// TIA Portal project "btvn" (V14)

(* hardware
DEVICE "S7-1200 station_1"  S7-1200 Station
   slot 0: "Rack_0"  S7-1200 Rack  Rack  V1.0
   slot 1: "PLC_1"  CPU 1214C DC/DC/DC  6ES7 214-1AG40-0XB0  V4.2
*)

// ===== PLC "PLC_1"  CPU 1214C DC/DC/DC =====

VAR_GLOBAL   // PLC tag table "Default tag table"
   "button1" AT %I0.1 : Bool;
   "button2" AT %I0.2 : Bool;
   "start" AT %I0.3 : Bool;
   "red_1" AT %Q0.2 : Bool;
   "red_2" AT %Q0.3 : Bool;
   "green_1" AT %Q0.0 : Bool;
   "green2" AT %Q0.1 : Bool;
   "reset" AT %I0.4 : Bool;
   "save1" AT %M1.0 : Bool;
   "save2" AT %M1.1 : Bool;
   "Start_button_" AT %M1.2 : Bool;
   "but1" AT %M0.0 : Bool;
   "den" AT %M0.1 : Bool;
END_VAR

ORGANIZATION_BLOCK "Main"   // OB1, LAD, ProgramCycle
TITLE = "Main Program Sweep (Cycle)"
{ S7_Optimized_Access := 'TRUE' }
VERSION : 0.1
   VAR_INPUT
      Initial_Call : Bool;   // Initial call of this OB
      Remanence : Bool;   // =True, if remanent data are available
   END_VAR
   VAR_TEMP
      Start_button : Bool;
   END_VAR
   VAR_TEMP   // added for the SCL form of the ladder/FBD networks
      _w1 : Bool;
   END_VAR
BEGIN

REGION Network 1
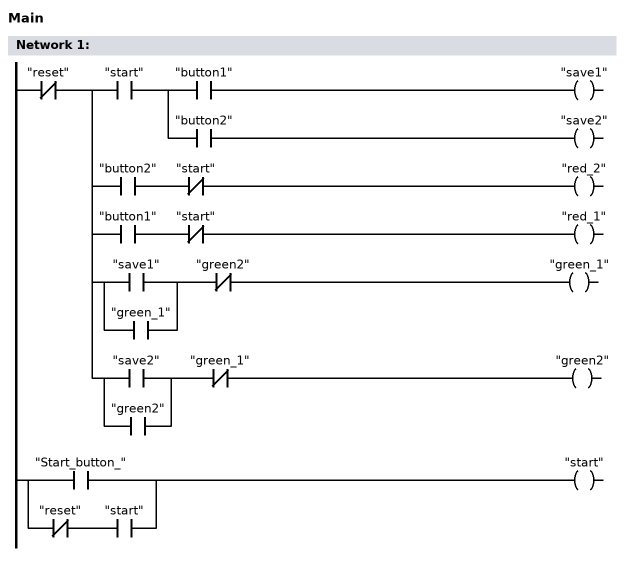
   RUNG wire#powerrail
      I_Contact( "reset" )
      wire#w1
      Contact( "start" )
      wire#w2
      Contact( "button1" )
      Coil( "save1" )
   END_RUNG
   RUNG wire#w2
      Contact( "button2" )
      Coil( "save2" )
   END_RUNG
   RUNG wire#w1
      Contact( "button2" )
      I_Contact( "start" )
      Coil( "red_2" )
   END_RUNG
   RUNG wire#w1
      Contact( "button1" )
      I_Contact( "start" )
      Coil( "red_1" )
   END_RUNG
   RUNG wire#w1
      Contact( "save1" )
      wire#w3
      I_Contact( "green2" )
      Coil( "green_1" )
   END_RUNG
   RUNG wire#w1
      Contact( "green_1" )
   END_RUNG wire#w3
   RUNG wire#w1
      Contact( "save2" )
      wire#w4
      I_Contact( "green_1" )
      Coil( "green2" )
   END_RUNG
   RUNG wire#w1
      Contact( "green2" )
   END_RUNG wire#w4
   RUNG wire#powerrail
      Contact( "Start_button_" )
      wire#w5
      Coil( "start" )
   END_RUNG
   RUNG wire#powerrail
      I_Contact( "reset" )
      Contact( "start" )
   END_RUNG wire#w5
   // the same network as SCL:
   #_w1 := NOT "reset" AND "start";
   "save1" := #_w1 AND "button1";
   "save2" := #_w1 AND "button2";
   "red_2" := NOT "reset" AND "button2" AND NOT "start";
   "red_1" := NOT "reset" AND "button1" AND NOT "start";
   "green_1" := NOT "reset" AND ("save1" OR "green_1") AND NOT "green2";
   "green2" := NOT "reset" AND ("save2" OR "green2") AND NOT "green_1";
   "start" := "Start_button_" OR (NOT "reset" AND "start");
END_REGION
END_ORGANIZATION_BLOCK